{attribute 'qualified_only'}
{attribute 'strict'}
TYPE MonitoringState :
(
	inactive := 0,
	railL,
	railR,
	railBoth,
	ownRail
);
END_TYPE

(* stored: Version 1.1.0.1, ProductVersion 3.1.4024.11
   DUT MonitoringState: Id {6792acb5-ae25-4296-be2e-45da1bc4e9d9} *)
